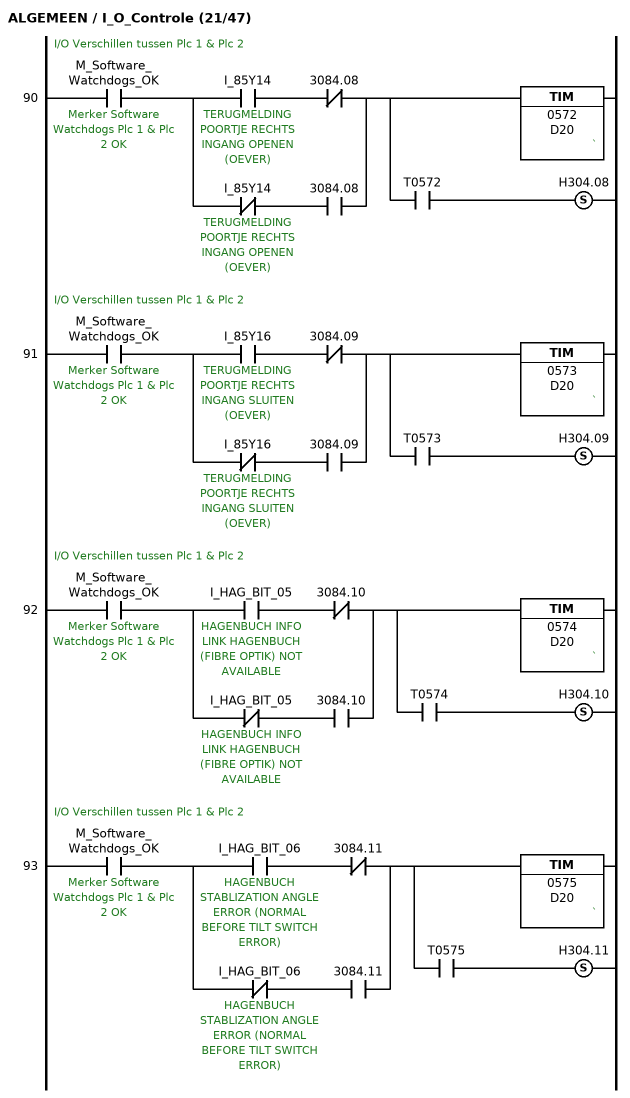
; [picture p229: ALGEMEEN / I_O_Controle, rungs 90-93]
; rung 90: I/O Verschillen tussen Plc 1 & Plc 2
LD M_Software_Watchdogs_OK  ; Merker Software Watchdogs Plc 1 & Plc 2 OK
LD I_85Y14  ; TERUGMELDING POORTJE RECHTS INGANG OPENEN (OEVER)
ANDNOT 3084.08
LDNOT I_85Y14  ; TERUGMELDING POORTJE RECHTS INGANG OPENEN (OEVER)
AND 3084.08
ORLD
ANDLD
TIM 0572 D20  ; `
AND T0572
SET H304.08
; rung 91: I/O Verschillen tussen Plc 1 & Plc 2
LD M_Software_Watchdogs_OK  ; Merker Software Watchdogs Plc 1 & Plc 2 OK
LD I_85Y16  ; TERUGMELDING POORTJE RECHTS INGANG SLUITEN (OEVER)
ANDNOT 3084.09
LDNOT I_85Y16  ; TERUGMELDING POORTJE RECHTS INGANG SLUITEN (OEVER)
AND 3084.09
ORLD
ANDLD
TIM 0573 D20  ; `
AND T0573
SET H304.09
; rung 92: I/O Verschillen tussen Plc 1 & Plc 2
LD M_Software_Watchdogs_OK  ; Merker Software Watchdogs Plc 1 & Plc 2 OK
LD I_HAG_BIT_05  ; HAGENBUCH INFO LINK HAGENBUCH (FIBRE OPTIK) NOT AVAILABLE
ANDNOT 3084.10
LDNOT I_HAG_BIT_05  ; HAGENBUCH INFO LINK HAGENBUCH (FIBRE OPTIK) NOT AVAILABLE
AND 3084.10
ORLD
ANDLD
TIM 0574 D20  ; `
AND T0574
SET H304.10
; rung 93: I/O Verschillen tussen Plc 1 & Plc 2
LD M_Software_Watchdogs_OK  ; Merker Software Watchdogs Plc 1 & Plc 2 OK
LD I_HAG_BIT_06  ; HAGENBUCH STABLIZATION ANGLE ERROR (NORMAL BEFORE TILT SWITCH ERROR)
ANDNOT 3084.11
LDNOT I_HAG_BIT_06  ; HAGENBUCH STABLIZATION ANGLE ERROR (NORMAL BEFORE TILT SWITCH ERROR)
AND 3084.11
ORLD
ANDLD
TIM 0575 D20  ; `
AND T0575
SET H304.11

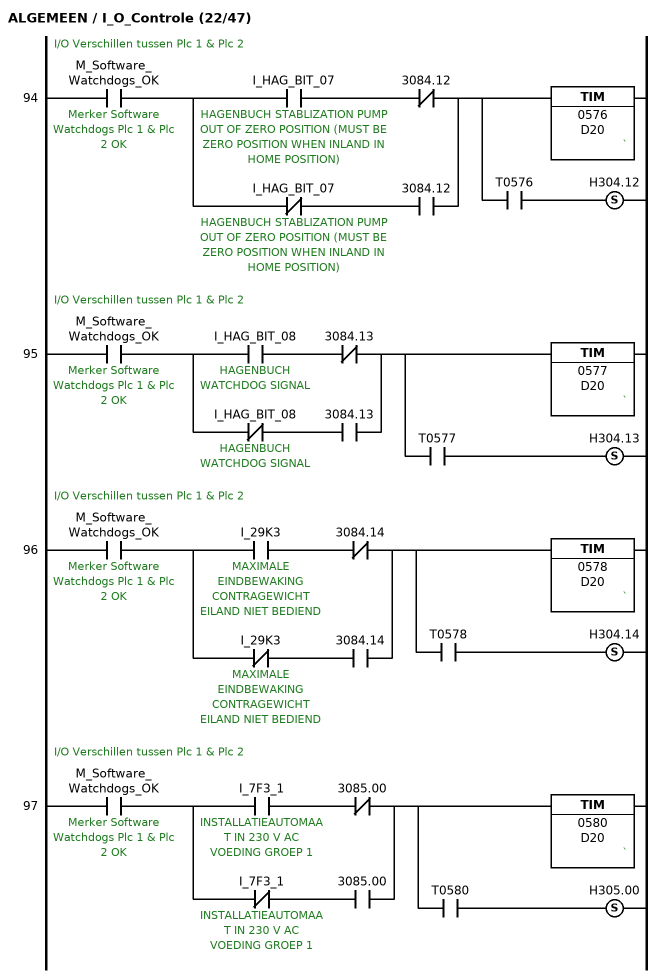
; rung 94: I/O Verschillen tussen Plc 1 & Plc 2
LD M_Software_Watchdogs_OK  ; Merker Software Watchdogs Plc 1 & Plc 2 OK
LD I_HAG_BIT_07  ; HAGENBUCH STABLIZATION PUMP OUT OF ZERO POSITION (MUST BE ZERO POSITION WHEN INLAND IN HOME POSITION)
ANDNOT 3084.12
LDNOT I_HAG_BIT_07  ; HAGENBUCH STABLIZATION PUMP OUT OF ZERO POSITION (MUST BE ZERO POSITION WHEN INLAND IN HOME POSITION)
AND 3084.12
ORLD
ANDLD
TIM 0576 D20  ; `
AND T0576
SET H304.12
; rung 95: I/O Verschillen tussen Plc 1 & Plc 2
LD M_Software_Watchdogs_OK  ; Merker Software Watchdogs Plc 1 & Plc 2 OK
LD I_HAG_BIT_08  ; HAGENBUCH WATCHDOG SIGNAL
ANDNOT 3084.13
LDNOT I_HAG_BIT_08  ; HAGENBUCH WATCHDOG SIGNAL
AND 3084.13
ORLD
ANDLD
TIM 0577 D20  ; `
AND T0577
SET H304.13
; rung 96: I/O Verschillen tussen Plc 1 & Plc 2
LD M_Software_Watchdogs_OK  ; Merker Software Watchdogs Plc 1 & Plc 2 OK
LD I_29K3  ; MAXIMALE EINDBEWAKING CONTRAGEWICHT EILAND NIET BEDIEND
ANDNOT 3084.14
LDNOT I_29K3  ; MAXIMALE EINDBEWAKING CONTRAGEWICHT EILAND NIET BEDIEND
AND 3084.14
ORLD
ANDLD
TIM 0578 D20  ; `
AND T0578
SET H304.14
; rung 97: I/O Verschillen tussen Plc 1 & Plc 2
LD M_Software_Watchdogs_OK  ; Merker Software Watchdogs Plc 1 & Plc 2 OK
LD I_7F3_1  ; INSTALLATIEAUTOMAAT IN 230 V AC VOEDING GROEP 1
ANDNOT 3085.00
LDNOT I_7F3_1  ; INSTALLATIEAUTOMAAT IN 230 V AC VOEDING GROEP 1
AND 3085.00
ORLD
ANDLD
TIM 0580 D20  ; `
AND T0580
SET H305.00

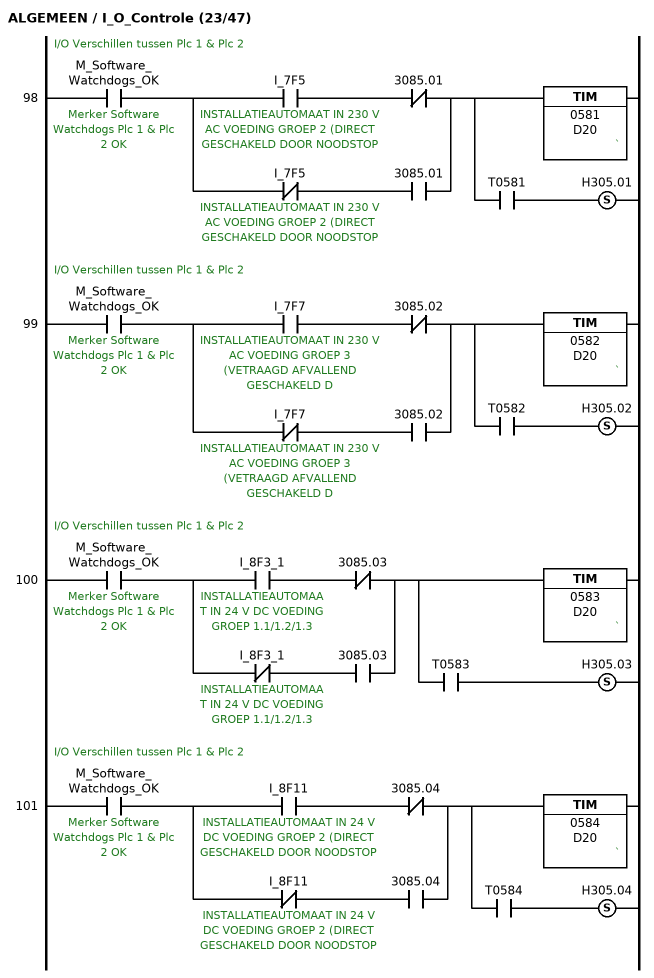
; rung 98: I/O Verschillen tussen Plc 1 & Plc 2
LD M_Software_Watchdogs_OK  ; Merker Software Watchdogs Plc 1 & Plc 2 OK
LD I_7F5  ; INSTALLATIEAUTOMAAT IN 230 V AC VOEDING GROEP 2 (DIRECT GESCHAKELD DOOR NOODSTOP
ANDNOT 3085.01
LDNOT I_7F5  ; INSTALLATIEAUTOMAAT IN 230 V AC VOEDING GROEP 2 (DIRECT GESCHAKELD DOOR NOODSTOP
AND 3085.01
ORLD
ANDLD
TIM 0581 D20  ; `
AND T0581
SET H305.01
; rung 99: I/O Verschillen tussen Plc 1 & Plc 2
LD M_Software_Watchdogs_OK  ; Merker Software Watchdogs Plc 1 & Plc 2 OK
LD I_7F7  ; INSTALLATIEAUTOMAAT IN 230 V AC VOEDING GROEP 3 (VETRAAGD AFVALLEND GESCHAKELD D
ANDNOT 3085.02
LDNOT I_7F7  ; INSTALLATIEAUTOMAAT IN 230 V AC VOEDING GROEP 3 (VETRAAGD AFVALLEND GESCHAKELD D
AND 3085.02
ORLD
ANDLD
TIM 0582 D20  ; `
AND T0582
SET H305.02
; rung 100: I/O Verschillen tussen Plc 1 & Plc 2
LD M_Software_Watchdogs_OK  ; Merker Software Watchdogs Plc 1 & Plc 2 OK
LD I_8F3_1  ; INSTALLATIEAUTOMAAT IN 24 V DC VOEDING GROEP 1.1/1.2/1.3
ANDNOT 3085.03
LDNOT I_8F3_1  ; INSTALLATIEAUTOMAAT IN 24 V DC VOEDING GROEP 1.1/1.2/1.3
AND 3085.03
ORLD
ANDLD
TIM 0583 D20  ; `
AND T0583
SET H305.03
; rung 101: I/O Verschillen tussen Plc 1 & Plc 2
LD M_Software_Watchdogs_OK  ; Merker Software Watchdogs Plc 1 & Plc 2 OK
LD I_8F11  ; INSTALLATIEAUTOMAAT IN 24 V DC VOEDING GROEP 2 (DIRECT GESCHAKELD DOOR NOODSTOP
ANDNOT 3085.04
LDNOT I_8F11  ; INSTALLATIEAUTOMAAT IN 24 V DC VOEDING GROEP 2 (DIRECT GESCHAKELD DOOR NOODSTOP
AND 3085.04
ORLD
ANDLD
TIM 0584 D20  ; `
AND T0584
SET H305.04

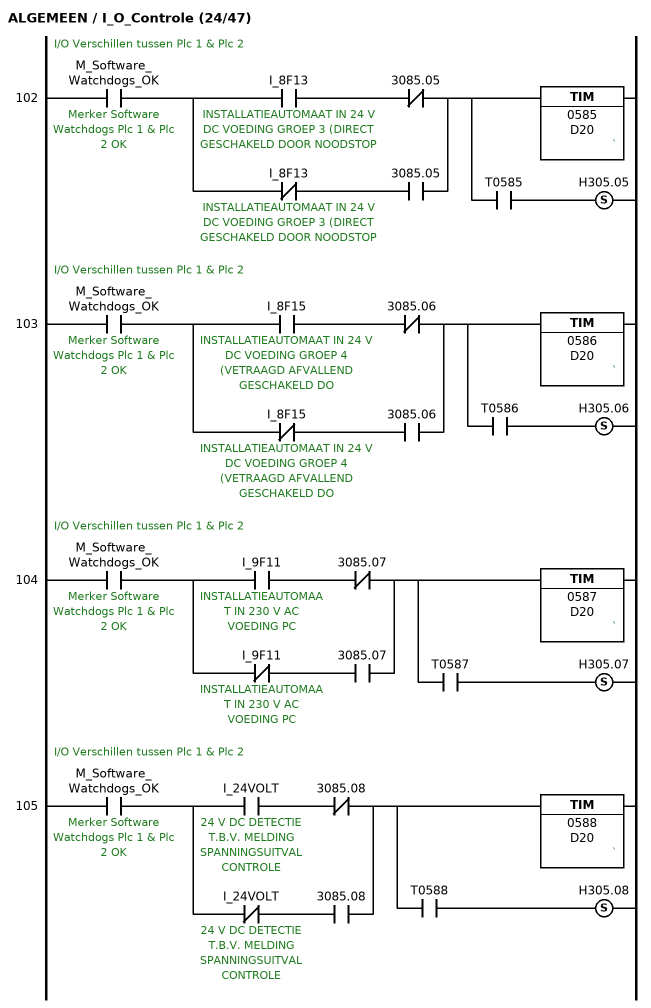
; rung 102: I/O Verschillen tussen Plc 1 & Plc 2
LD M_Software_Watchdogs_OK  ; Merker Software Watchdogs Plc 1 & Plc 2 OK
LD I_8F13  ; INSTALLATIEAUTOMAAT IN 24 V DC VOEDING GROEP 3 (DIRECT GESCHAKELD DOOR NOODSTOP
ANDNOT 3085.05
LDNOT I_8F13  ; INSTALLATIEAUTOMAAT IN 24 V DC VOEDING GROEP 3 (DIRECT GESCHAKELD DOOR NOODSTOP
AND 3085.05
ORLD
ANDLD
TIM 0585 D20  ; `
AND T0585
SET H305.05
; rung 103: I/O Verschillen tussen Plc 1 & Plc 2
LD M_Software_Watchdogs_OK  ; Merker Software Watchdogs Plc 1 & Plc 2 OK
LD I_8F15  ; INSTALLATIEAUTOMAAT IN 24 V DC VOEDING GROEP 4 (VETRAAGD AFVALLEND GESCHAKELD DO
ANDNOT 3085.06
LDNOT I_8F15  ; INSTALLATIEAUTOMAAT IN 24 V DC VOEDING GROEP 4 (VETRAAGD AFVALLEND GESCHAKELD DO
AND 3085.06
ORLD
ANDLD
TIM 0586 D20  ; `
AND T0586
SET H305.06
; rung 104: I/O Verschillen tussen Plc 1 & Plc 2
LD M_Software_Watchdogs_OK  ; Merker Software Watchdogs Plc 1 & Plc 2 OK
LD I_9F11  ; INSTALLATIEAUTOMAAT IN 230 V AC VOEDING PC
ANDNOT 3085.07
LDNOT I_9F11  ; INSTALLATIEAUTOMAAT IN 230 V AC VOEDING PC
AND 3085.07
ORLD
ANDLD
TIM 0587 D20  ; `
AND T0587
SET H305.07
; rung 105: I/O Verschillen tussen Plc 1 & Plc 2
LD M_Software_Watchdogs_OK  ; Merker Software Watchdogs Plc 1 & Plc 2 OK
LD I_24VOLT  ; 24 V DC DETECTIE T.B.V. MELDING SPANNINGSUITVAL CONTROLE
ANDNOT 3085.08
LDNOT I_24VOLT  ; 24 V DC DETECTIE T.B.V. MELDING SPANNINGSUITVAL CONTROLE
AND 3085.08
ORLD
ANDLD
TIM 0588 D20  ; `
AND T0588
SET H305.08

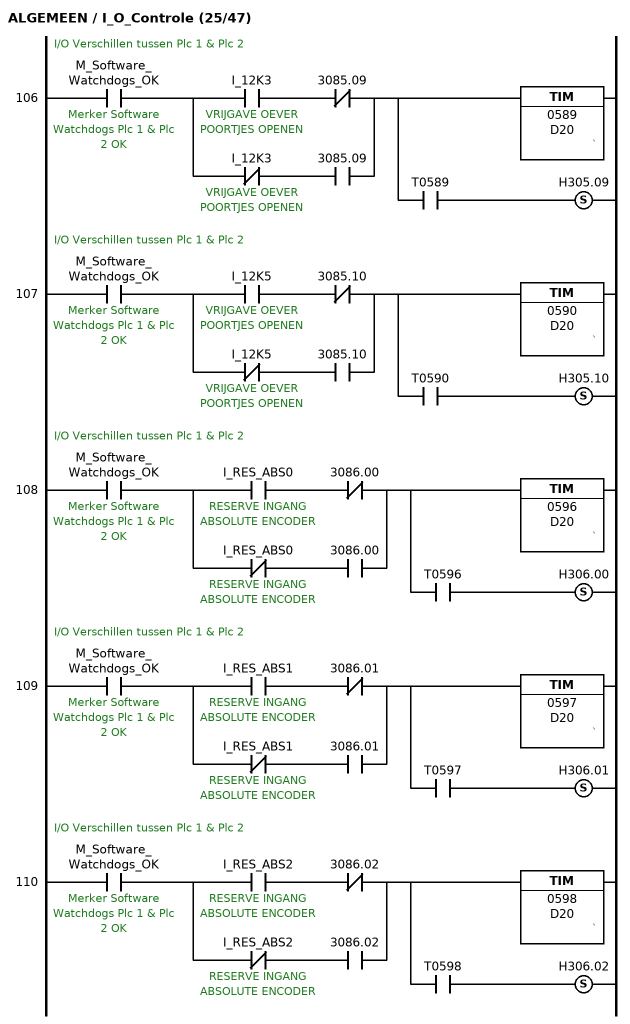
; rung 106: I/O Verschillen tussen Plc 1 & Plc 2
LD M_Software_Watchdogs_OK  ; Merker Software Watchdogs Plc 1 & Plc 2 OK
LD I_12K3  ; VRIJGAVE OEVER POORTJES OPENEN
ANDNOT 3085.09
LDNOT I_12K3  ; VRIJGAVE OEVER POORTJES OPENEN
AND 3085.09
ORLD
ANDLD
TIM 0589 D20  ; `
AND T0589
SET H305.09
; rung 107: I/O Verschillen tussen Plc 1 & Plc 2
LD M_Software_Watchdogs_OK  ; Merker Software Watchdogs Plc 1 & Plc 2 OK
LD I_12K5  ; VRIJGAVE OEVER POORTJES OPENEN
ANDNOT 3085.10
LDNOT I_12K5  ; VRIJGAVE OEVER POORTJES OPENEN
AND 3085.10
ORLD
ANDLD
TIM 0590 D20  ; `
AND T0590
SET H305.10
; rung 108: I/O Verschillen tussen Plc 1 & Plc 2
LD M_Software_Watchdogs_OK  ; Merker Software Watchdogs Plc 1 & Plc 2 OK
LD I_RES_ABS0  ; RESERVE INGANG ABSOLUTE ENCODER
ANDNOT 3086.00
LDNOT I_RES_ABS0  ; RESERVE INGANG ABSOLUTE ENCODER
AND 3086.00
ORLD
ANDLD
TIM 0596 D20  ; `
AND T0596
SET H306.00
; rung 109: I/O Verschillen tussen Plc 1 & Plc 2
LD M_Software_Watchdogs_OK  ; Merker Software Watchdogs Plc 1 & Plc 2 OK
LD I_RES_ABS1  ; RESERVE INGANG ABSOLUTE ENCODER
ANDNOT 3086.01
LDNOT I_RES_ABS1  ; RESERVE INGANG ABSOLUTE ENCODER
AND 3086.01
ORLD
ANDLD
TIM 0597 D20  ; `
AND T0597
SET H306.01
; rung 110: I/O Verschillen tussen Plc 1 & Plc 2
LD M_Software_Watchdogs_OK  ; Merker Software Watchdogs Plc 1 & Plc 2 OK
LD I_RES_ABS2  ; RESERVE INGANG ABSOLUTE ENCODER
ANDNOT 3086.02
LDNOT I_RES_ABS2  ; RESERVE INGANG ABSOLUTE ENCODER
AND 3086.02
ORLD
ANDLD
TIM 0598 D20  ; `
AND T0598
SET H306.02

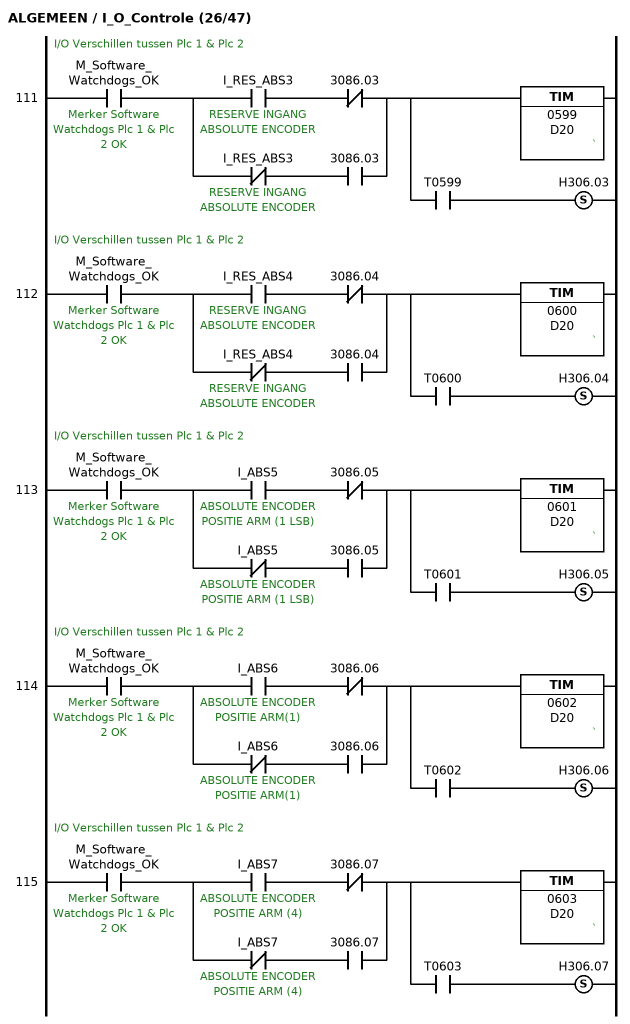
; rung 111: I/O Verschillen tussen Plc 1 & Plc 2
LD M_Software_Watchdogs_OK  ; Merker Software Watchdogs Plc 1 & Plc 2 OK
LD I_RES_ABS3  ; RESERVE INGANG ABSOLUTE ENCODER
ANDNOT 3086.03
LDNOT I_RES_ABS3  ; RESERVE INGANG ABSOLUTE ENCODER
AND 3086.03
ORLD
ANDLD
TIM 0599 D20  ; `
AND T0599
SET H306.03
; rung 112: I/O Verschillen tussen Plc 1 & Plc 2
LD M_Software_Watchdogs_OK  ; Merker Software Watchdogs Plc 1 & Plc 2 OK
LD I_RES_ABS4  ; RESERVE INGANG ABSOLUTE ENCODER
ANDNOT 3086.04
LDNOT I_RES_ABS4  ; RESERVE INGANG ABSOLUTE ENCODER
AND 3086.04
ORLD
ANDLD
TIM 0600 D20  ; `
AND T0600
SET H306.04
; rung 113: I/O Verschillen tussen Plc 1 & Plc 2
LD M_Software_Watchdogs_OK  ; Merker Software Watchdogs Plc 1 & Plc 2 OK
LD I_ABS5  ; ABSOLUTE ENCODER POSITIE ARM (1 LSB)
ANDNOT 3086.05
LDNOT I_ABS5  ; ABSOLUTE ENCODER POSITIE ARM (1 LSB)
AND 3086.05
ORLD
ANDLD
TIM 0601 D20  ; `
AND T0601
SET H306.05
; rung 114: I/O Verschillen tussen Plc 1 & Plc 2
LD M_Software_Watchdogs_OK  ; Merker Software Watchdogs Plc 1 & Plc 2 OK
LD I_ABS6  ; ABSOLUTE ENCODER POSITIE ARM(1)
ANDNOT 3086.06
LDNOT I_ABS6  ; ABSOLUTE ENCODER POSITIE ARM(1)
AND 3086.06
ORLD
ANDLD
TIM 0602 D20  ; `
AND T0602
SET H306.06
; rung 115: I/O Verschillen tussen Plc 1 & Plc 2
LD M_Software_Watchdogs_OK  ; Merker Software Watchdogs Plc 1 & Plc 2 OK
LD I_ABS7  ; ABSOLUTE ENCODER POSITIE ARM (4)
ANDNOT 3086.07
LDNOT I_ABS7  ; ABSOLUTE ENCODER POSITIE ARM (4)
AND 3086.07
ORLD
ANDLD
TIM 0603 D20  ; `
AND T0603
SET H306.07

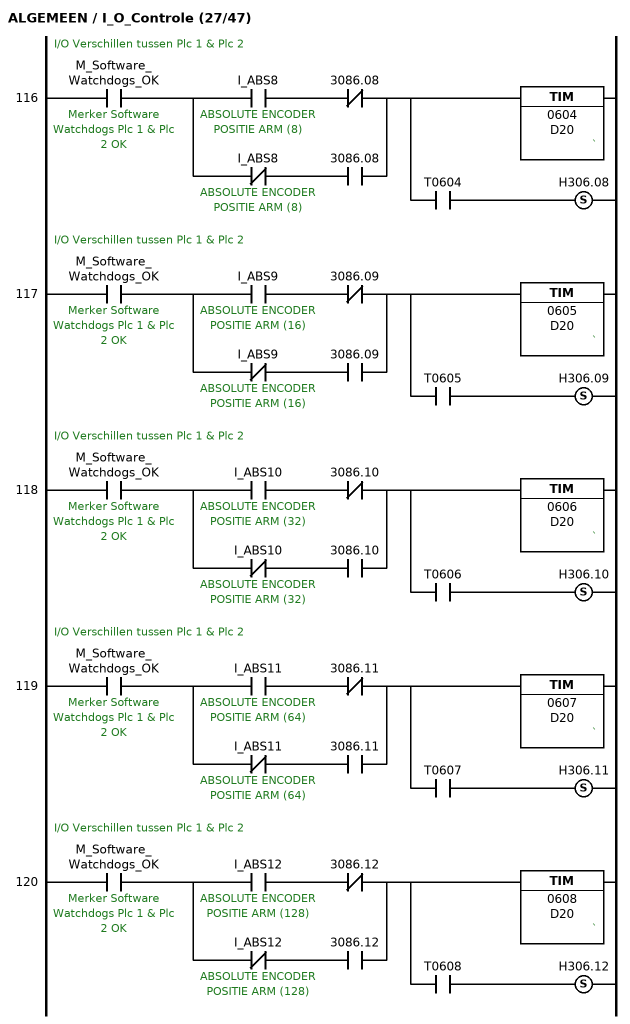
; rung 116: I/O Verschillen tussen Plc 1 & Plc 2
LD M_Software_Watchdogs_OK  ; Merker Software Watchdogs Plc 1 & Plc 2 OK
LD I_ABS8  ; ABSOLUTE ENCODER POSITIE ARM (8)
ANDNOT 3086.08
LDNOT I_ABS8  ; ABSOLUTE ENCODER POSITIE ARM (8)
AND 3086.08
ORLD
ANDLD
TIM 0604 D20  ; `
AND T0604
SET H306.08
; rung 117: I/O Verschillen tussen Plc 1 & Plc 2
LD M_Software_Watchdogs_OK  ; Merker Software Watchdogs Plc 1 & Plc 2 OK
LD I_ABS9  ; ABSOLUTE ENCODER POSITIE ARM (16)
ANDNOT 3086.09
LDNOT I_ABS9  ; ABSOLUTE ENCODER POSITIE ARM (16)
AND 3086.09
ORLD
ANDLD
TIM 0605 D20  ; `
AND T0605
SET H306.09
; rung 118: I/O Verschillen tussen Plc 1 & Plc 2
LD M_Software_Watchdogs_OK  ; Merker Software Watchdogs Plc 1 & Plc 2 OK
LD I_ABS10  ; ABSOLUTE ENCODER POSITIE ARM (32)
ANDNOT 3086.10
LDNOT I_ABS10  ; ABSOLUTE ENCODER POSITIE ARM (32)
AND 3086.10
ORLD
ANDLD
TIM 0606 D20  ; `
AND T0606
SET H306.10
; rung 119: I/O Verschillen tussen Plc 1 & Plc 2
LD M_Software_Watchdogs_OK  ; Merker Software Watchdogs Plc 1 & Plc 2 OK
LD I_ABS11  ; ABSOLUTE ENCODER POSITIE ARM (64)
ANDNOT 3086.11
LDNOT I_ABS11  ; ABSOLUTE ENCODER POSITIE ARM (64)
AND 3086.11
ORLD
ANDLD
TIM 0607 D20  ; `
AND T0607
SET H306.11
; rung 120: I/O Verschillen tussen Plc 1 & Plc 2
LD M_Software_Watchdogs_OK  ; Merker Software Watchdogs Plc 1 & Plc 2 OK
LD I_ABS12  ; ABSOLUTE ENCODER POSITIE ARM (128)
ANDNOT 3086.12
LDNOT I_ABS12  ; ABSOLUTE ENCODER POSITIE ARM (128)
AND 3086.12
ORLD
ANDLD
TIM 0608 D20  ; `
AND T0608
SET H306.12

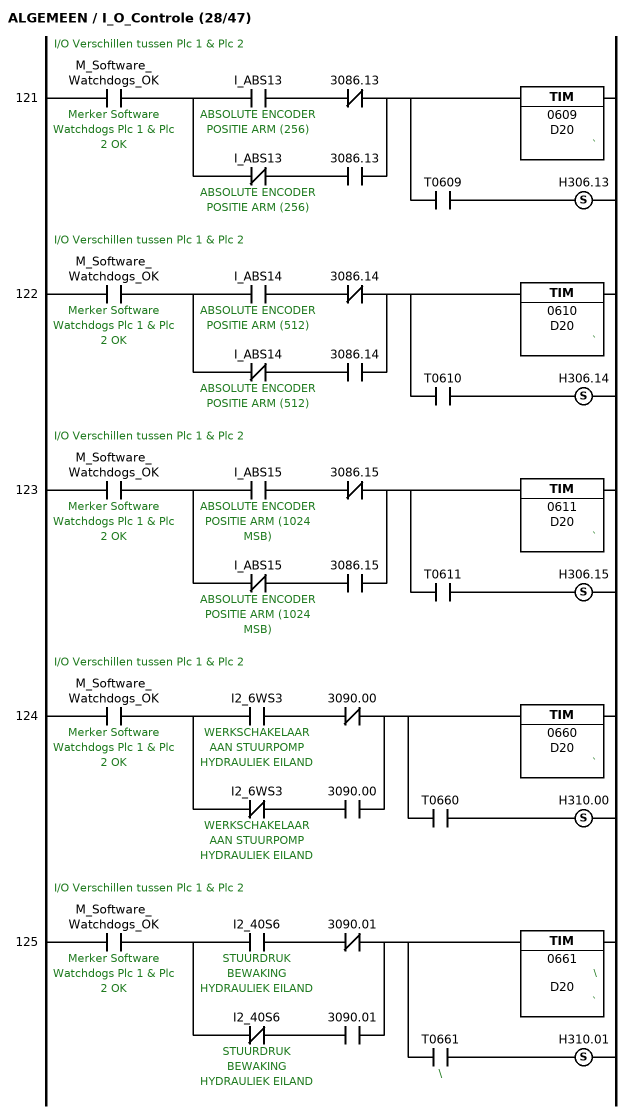
; rung 121: I/O Verschillen tussen Plc 1 & Plc 2
LD M_Software_Watchdogs_OK  ; Merker Software Watchdogs Plc 1 & Plc 2 OK
LD I_ABS13  ; ABSOLUTE ENCODER POSITIE ARM (256)
ANDNOT 3086.13
LDNOT I_ABS13  ; ABSOLUTE ENCODER POSITIE ARM (256)
AND 3086.13
ORLD
ANDLD
TIM 0609 D20  ; `
AND T0609
SET H306.13
; rung 122: I/O Verschillen tussen Plc 1 & Plc 2
LD M_Software_Watchdogs_OK  ; Merker Software Watchdogs Plc 1 & Plc 2 OK
LD I_ABS14  ; ABSOLUTE ENCODER POSITIE ARM (512)
ANDNOT 3086.14
LDNOT I_ABS14  ; ABSOLUTE ENCODER POSITIE ARM (512)
AND 3086.14
ORLD
ANDLD
TIM 0610 D20  ; `
AND T0610
SET H306.14
; rung 123: I/O Verschillen tussen Plc 1 & Plc 2
LD M_Software_Watchdogs_OK  ; Merker Software Watchdogs Plc 1 & Plc 2 OK
LD I_ABS15  ; ABSOLUTE ENCODER POSITIE ARM (1024 MSB)
ANDNOT 3086.15
LDNOT I_ABS15  ; ABSOLUTE ENCODER POSITIE ARM (1024 MSB)
AND 3086.15
ORLD
ANDLD
TIM 0611 D20  ; `
AND T0611
SET H306.15
; rung 124: I/O Verschillen tussen Plc 1 & Plc 2
LD M_Software_Watchdogs_OK  ; Merker Software Watchdogs Plc 1 & Plc 2 OK
LD I2_6WS3  ; WERKSCHAKELAAR AAN STUURPOMP HYDRAULIEK EILAND
ANDNOT 3090.00
LDNOT I2_6WS3  ; WERKSCHAKELAAR AAN STUURPOMP HYDRAULIEK EILAND
AND 3090.00
ORLD
ANDLD
TIM 0660 D20  ; `
AND T0660
SET H310.00
; rung 125: I/O Verschillen tussen Plc 1 & Plc 2
LD M_Software_Watchdogs_OK  ; Merker Software Watchdogs Plc 1 & Plc 2 OK
LD I2_40S6  ; STUURDRUK BEWAKING HYDRAULIEK EILAND
ANDNOT 3090.01
LDNOT I2_40S6  ; STUURDRUK BEWAKING HYDRAULIEK EILAND
AND 3090.01
ORLD
ANDLD
TIM 0661 D20  ; `, \
AND T0661  ; \
SET H310.01

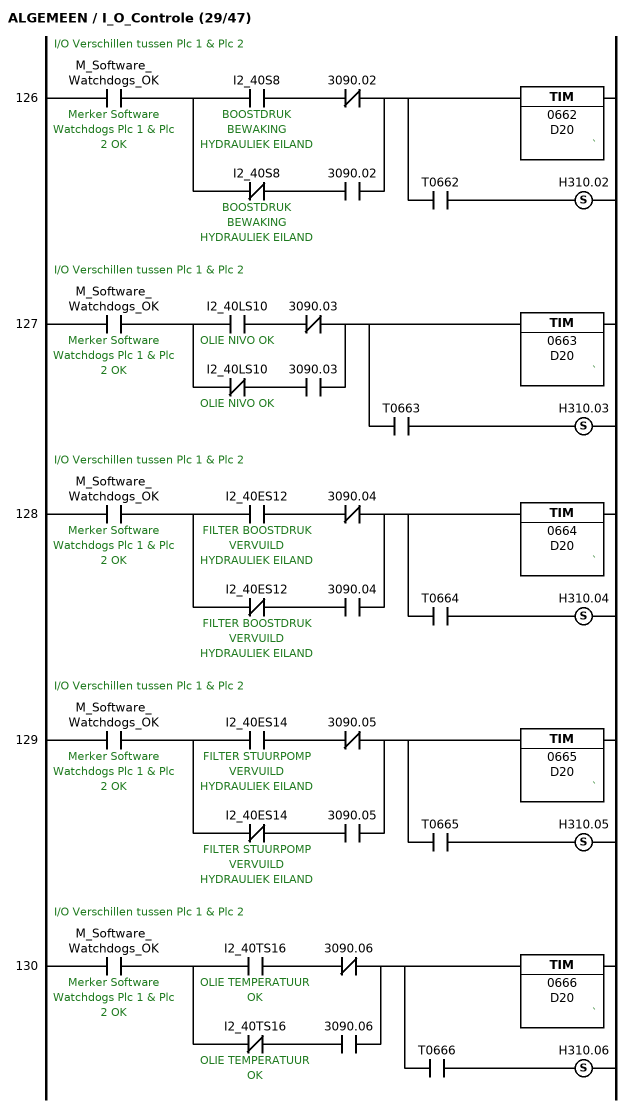
; rung 126: I/O Verschillen tussen Plc 1 & Plc 2
LD M_Software_Watchdogs_OK  ; Merker Software Watchdogs Plc 1 & Plc 2 OK
LD I2_40S8  ; BOOSTDRUK BEWAKING HYDRAULIEK EILAND
ANDNOT 3090.02
LDNOT I2_40S8  ; BOOSTDRUK BEWAKING HYDRAULIEK EILAND
AND 3090.02
ORLD
ANDLD
TIM 0662 D20  ; `
AND T0662
SET H310.02
; rung 127: I/O Verschillen tussen Plc 1 & Plc 2
LD M_Software_Watchdogs_OK  ; Merker Software Watchdogs Plc 1 & Plc 2 OK
LD I2_40LS10  ; OLIE NIVO OK
ANDNOT 3090.03
LDNOT I2_40LS10  ; OLIE NIVO OK
AND 3090.03
ORLD
ANDLD
TIM 0663 D20  ; `
AND T0663
SET H310.03
; rung 128: I/O Verschillen tussen Plc 1 & Plc 2
LD M_Software_Watchdogs_OK  ; Merker Software Watchdogs Plc 1 & Plc 2 OK
LD I2_40ES12  ; FILTER BOOSTDRUK VERVUILD HYDRAULIEK EILAND
ANDNOT 3090.04
LDNOT I2_40ES12  ; FILTER BOOSTDRUK VERVUILD HYDRAULIEK EILAND
AND 3090.04
ORLD
ANDLD
TIM 0664 D20  ; `
AND T0664
SET H310.04
; rung 129: I/O Verschillen tussen Plc 1 & Plc 2
LD M_Software_Watchdogs_OK  ; Merker Software Watchdogs Plc 1 & Plc 2 OK
LD I2_40ES14  ; FILTER STUURPOMP VERVUILD HYDRAULIEK EILAND
ANDNOT 3090.05
LDNOT I2_40ES14  ; FILTER STUURPOMP VERVUILD HYDRAULIEK EILAND
AND 3090.05
ORLD
ANDLD
TIM 0665 D20  ; `
AND T0665
SET H310.05
; rung 130: I/O Verschillen tussen Plc 1 & Plc 2
LD M_Software_Watchdogs_OK  ; Merker Software Watchdogs Plc 1 & Plc 2 OK
LD I2_40TS16  ; OLIE TEMPERATUUR OK
ANDNOT 3090.06
LDNOT I2_40TS16  ; OLIE TEMPERATUUR OK
AND 3090.06
ORLD
ANDLD
TIM 0666 D20  ; `
AND T0666
SET H310.06

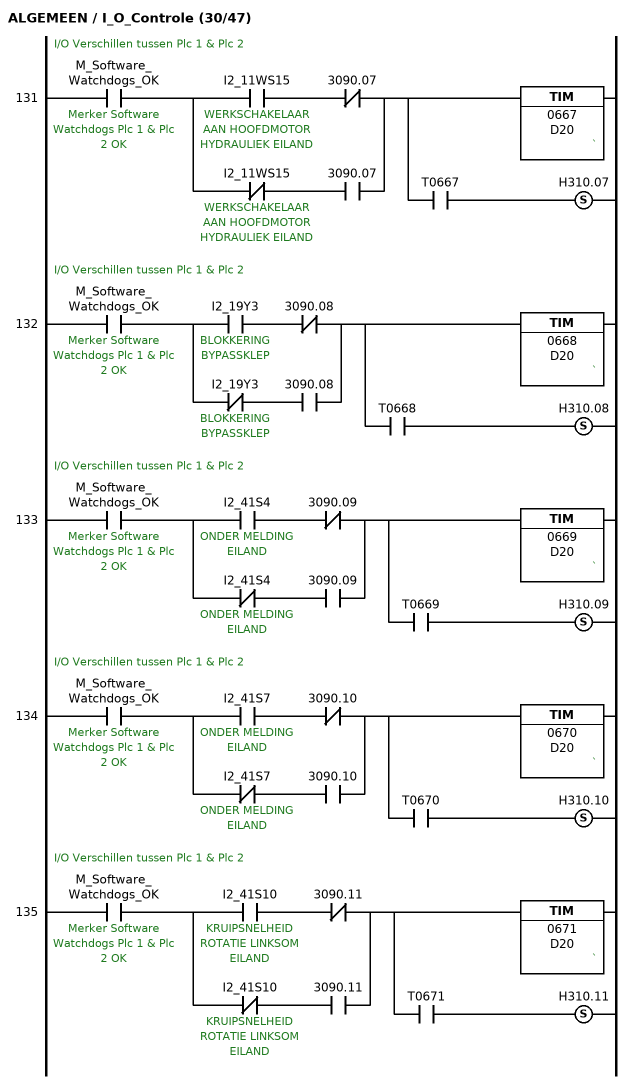
; rung 131: I/O Verschillen tussen Plc 1 & Plc 2
LD M_Software_Watchdogs_OK  ; Merker Software Watchdogs Plc 1 & Plc 2 OK
LD I2_11WS15  ; WERKSCHAKELAAR AAN HOOFDMOTOR HYDRAULIEK EILAND
ANDNOT 3090.07
LDNOT I2_11WS15  ; WERKSCHAKELAAR AAN HOOFDMOTOR HYDRAULIEK EILAND
AND 3090.07
ORLD
ANDLD
TIM 0667 D20  ; `
AND T0667
SET H310.07
; rung 132: I/O Verschillen tussen Plc 1 & Plc 2
LD M_Software_Watchdogs_OK  ; Merker Software Watchdogs Plc 1 & Plc 2 OK
LD I2_19Y3  ; BLOKKERING BYPASSKLEP
ANDNOT 3090.08
LDNOT I2_19Y3  ; BLOKKERING BYPASSKLEP
AND 3090.08
ORLD
ANDLD
TIM 0668 D20  ; `
AND T0668
SET H310.08
; rung 133: I/O Verschillen tussen Plc 1 & Plc 2
LD M_Software_Watchdogs_OK  ; Merker Software Watchdogs Plc 1 & Plc 2 OK
LD I2_41S4  ; ONDER MELDING EILAND
ANDNOT 3090.09
LDNOT I2_41S4  ; ONDER MELDING EILAND
AND 3090.09
ORLD
ANDLD
TIM 0669 D20  ; `
AND T0669
SET H310.09
; rung 134: I/O Verschillen tussen Plc 1 & Plc 2
LD M_Software_Watchdogs_OK  ; Merker Software Watchdogs Plc 1 & Plc 2 OK
LD I2_41S7  ; ONDER MELDING EILAND
ANDNOT 3090.10
LDNOT I2_41S7  ; ONDER MELDING EILAND
AND 3090.10
ORLD
ANDLD
TIM 0670 D20  ; `
AND T0670
SET H310.10
; rung 135: I/O Verschillen tussen Plc 1 & Plc 2
LD M_Software_Watchdogs_OK  ; Merker Software Watchdogs Plc 1 & Plc 2 OK
LD I2_41S10  ; KRUIPSNELHEID ROTATIE LINKSOM EILAND
ANDNOT 3090.11
LDNOT I2_41S10  ; KRUIPSNELHEID ROTATIE LINKSOM EILAND
AND 3090.11
ORLD
ANDLD
TIM 0671 D20  ; `
AND T0671
SET H310.11

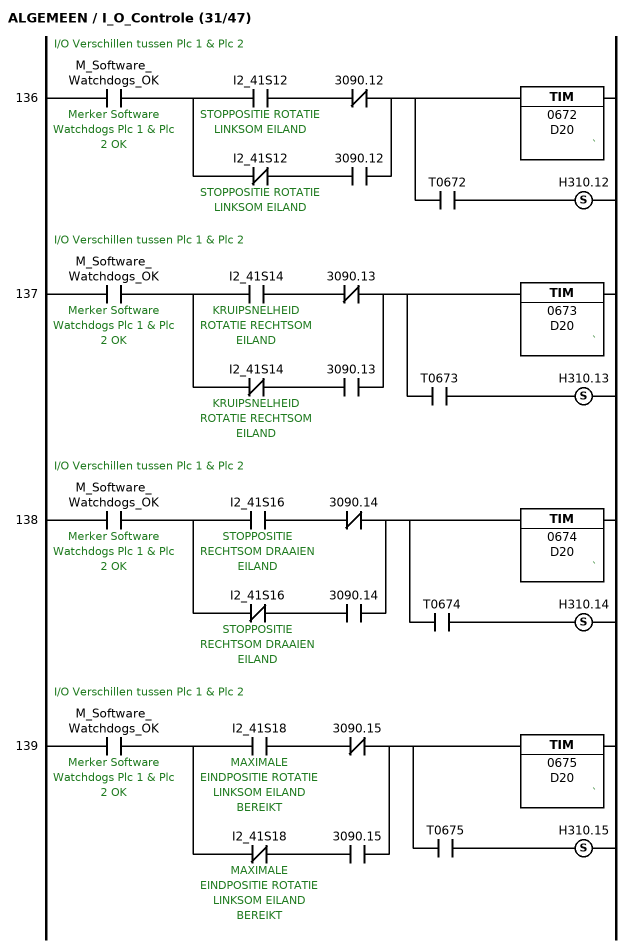
; rung 136: I/O Verschillen tussen Plc 1 & Plc 2
LD M_Software_Watchdogs_OK  ; Merker Software Watchdogs Plc 1 & Plc 2 OK
LD I2_41S12  ; STOPPOSITIE ROTATIE LINKSOM EILAND
ANDNOT 3090.12
LDNOT I2_41S12  ; STOPPOSITIE ROTATIE LINKSOM EILAND
AND 3090.12
ORLD
ANDLD
TIM 0672 D20  ; `
AND T0672
SET H310.12
; rung 137: I/O Verschillen tussen Plc 1 & Plc 2
LD M_Software_Watchdogs_OK  ; Merker Software Watchdogs Plc 1 & Plc 2 OK
LD I2_41S14  ; KRUIPSNELHEID ROTATIE RECHTSOM EILAND
ANDNOT 3090.13
LDNOT I2_41S14  ; KRUIPSNELHEID ROTATIE RECHTSOM EILAND
AND 3090.13
ORLD
ANDLD
TIM 0673 D20  ; `
AND T0673
SET H310.13
; rung 138: I/O Verschillen tussen Plc 1 & Plc 2
LD M_Software_Watchdogs_OK  ; Merker Software Watchdogs Plc 1 & Plc 2 OK
LD I2_41S16  ; STOPPOSITIE RECHTSOM DRAAIEN EILAND
ANDNOT 3090.14
LDNOT I2_41S16  ; STOPPOSITIE RECHTSOM DRAAIEN EILAND
AND 3090.14
ORLD
ANDLD
TIM 0674 D20  ; `
AND T0674
SET H310.14
; rung 139: I/O Verschillen tussen Plc 1 & Plc 2
LD M_Software_Watchdogs_OK  ; Merker Software Watchdogs Plc 1 & Plc 2 OK
LD I2_41S18  ; MAXIMALE EINDPOSITIE ROTATIE LINKSOM EILAND BEREIKT
ANDNOT 3090.15
LDNOT I2_41S18  ; MAXIMALE EINDPOSITIE ROTATIE LINKSOM EILAND BEREIKT
AND 3090.15
ORLD
ANDLD
TIM 0675 D20  ; `
AND T0675
SET H310.15

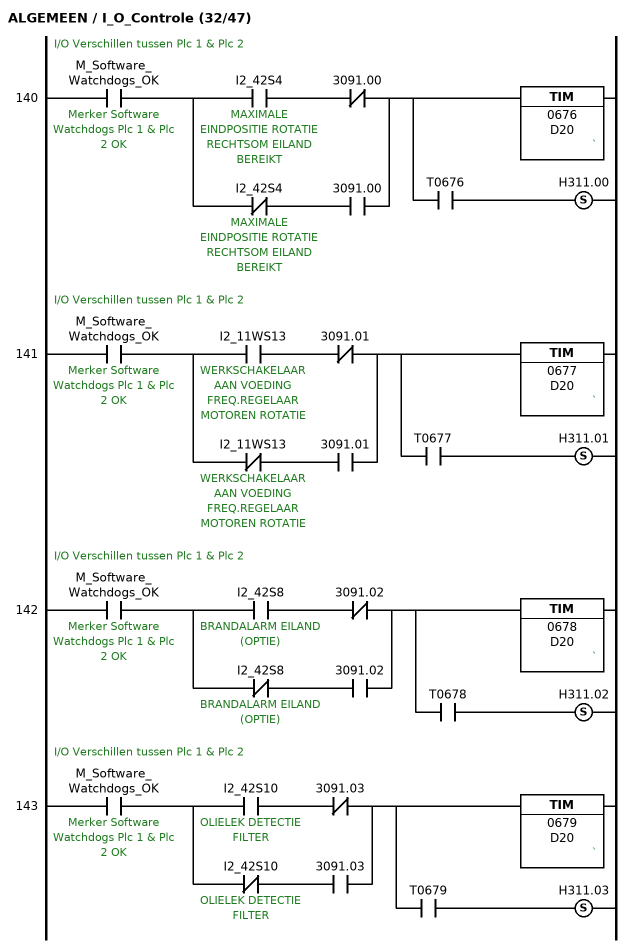
; rung 140: I/O Verschillen tussen Plc 1 & Plc 2
LD M_Software_Watchdogs_OK  ; Merker Software Watchdogs Plc 1 & Plc 2 OK
LD I2_42S4  ; MAXIMALE EINDPOSITIE ROTATIE RECHTSOM EILAND BEREIKT
ANDNOT 3091.00
LDNOT I2_42S4  ; MAXIMALE EINDPOSITIE ROTATIE RECHTSOM EILAND BEREIKT
AND 3091.00
ORLD
ANDLD
TIM 0676 D20  ; `
AND T0676
SET H311.00
; rung 141: I/O Verschillen tussen Plc 1 & Plc 2
LD M_Software_Watchdogs_OK  ; Merker Software Watchdogs Plc 1 & Plc 2 OK
LD I2_11WS13  ; WERKSCHAKELAAR AAN VOEDING FREQ.REGELAAR MOTOREN ROTATIE
ANDNOT 3091.01
LDNOT I2_11WS13  ; WERKSCHAKELAAR AAN VOEDING FREQ.REGELAAR MOTOREN ROTATIE
AND 3091.01
ORLD
ANDLD
TIM 0677 D20  ; `
AND T0677
SET H311.01
; rung 142: I/O Verschillen tussen Plc 1 & Plc 2
LD M_Software_Watchdogs_OK  ; Merker Software Watchdogs Plc 1 & Plc 2 OK
LD I2_42S8  ; BRANDALARM EILAND (OPTIE)
ANDNOT 3091.02
LDNOT I2_42S8  ; BRANDALARM EILAND (OPTIE)
AND 3091.02
ORLD
ANDLD
TIM 0678 D20  ; `
AND T0678
SET H311.02
; rung 143: I/O Verschillen tussen Plc 1 & Plc 2
LD M_Software_Watchdogs_OK  ; Merker Software Watchdogs Plc 1 & Plc 2 OK
LD I2_42S10  ; OLIELEK DETECTIE FILTER
ANDNOT 3091.03
LDNOT I2_42S10  ; OLIELEK DETECTIE FILTER
AND 3091.03
ORLD
ANDLD
TIM 0679 D20  ; `
AND T0679
SET H311.03

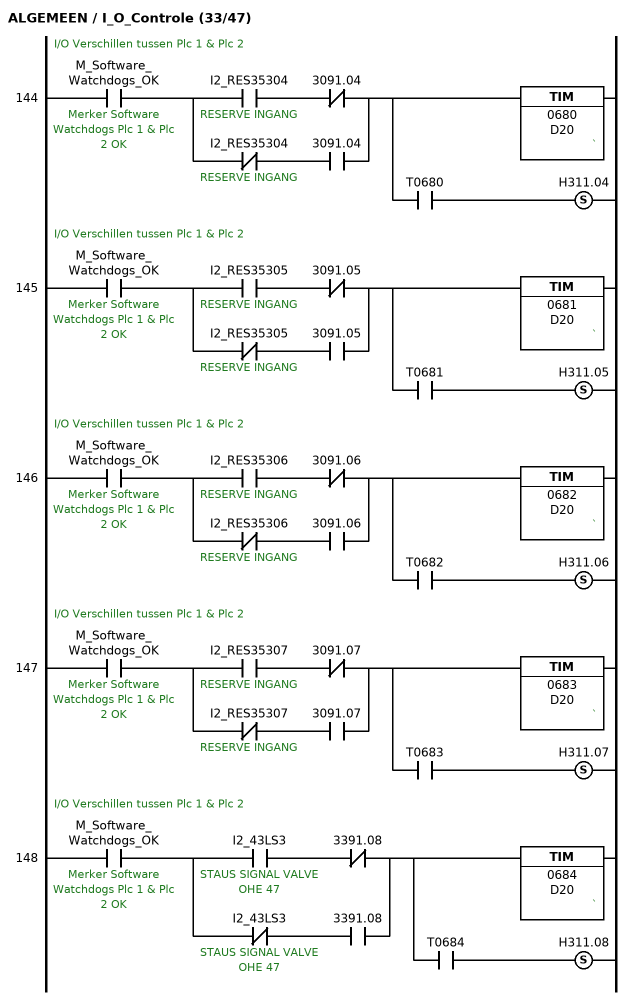
; rung 144: I/O Verschillen tussen Plc 1 & Plc 2
LD M_Software_Watchdogs_OK  ; Merker Software Watchdogs Plc 1 & Plc 2 OK
LD I2_RES35304  ; RESERVE INGANG
ANDNOT 3091.04
LDNOT I2_RES35304  ; RESERVE INGANG
AND 3091.04
ORLD
ANDLD
TIM 0680 D20  ; `
AND T0680
SET H311.04
; rung 145: I/O Verschillen tussen Plc 1 & Plc 2
LD M_Software_Watchdogs_OK  ; Merker Software Watchdogs Plc 1 & Plc 2 OK
LD I2_RES35305  ; RESERVE INGANG
ANDNOT 3091.05
LDNOT I2_RES35305  ; RESERVE INGANG
AND 3091.05
ORLD
ANDLD
TIM 0681 D20  ; `
AND T0681
SET H311.05
; rung 146: I/O Verschillen tussen Plc 1 & Plc 2
LD M_Software_Watchdogs_OK  ; Merker Software Watchdogs Plc 1 & Plc 2 OK
LD I2_RES35306  ; RESERVE INGANG
ANDNOT 3091.06
LDNOT I2_RES35306  ; RESERVE INGANG
AND 3091.06
ORLD
ANDLD
TIM 0682 D20  ; `
AND T0682
SET H311.06
; rung 147: I/O Verschillen tussen Plc 1 & Plc 2
LD M_Software_Watchdogs_OK  ; Merker Software Watchdogs Plc 1 & Plc 2 OK
LD I2_RES35307  ; RESERVE INGANG
ANDNOT 3091.07
LDNOT I2_RES35307  ; RESERVE INGANG
AND 3091.07
ORLD
ANDLD
TIM 0683 D20  ; `
AND T0683
SET H311.07
; rung 148: I/O Verschillen tussen Plc 1 & Plc 2
LD M_Software_Watchdogs_OK  ; Merker Software Watchdogs Plc 1 & Plc 2 OK
LD I2_43LS3  ; STAUS SIGNAL VALVE OHE 47
ANDNOT 3391.08
LDNOT I2_43LS3  ; STAUS SIGNAL VALVE OHE 47
AND 3391.08
ORLD
ANDLD
TIM 0684 D20  ; `
AND T0684
SET H311.08

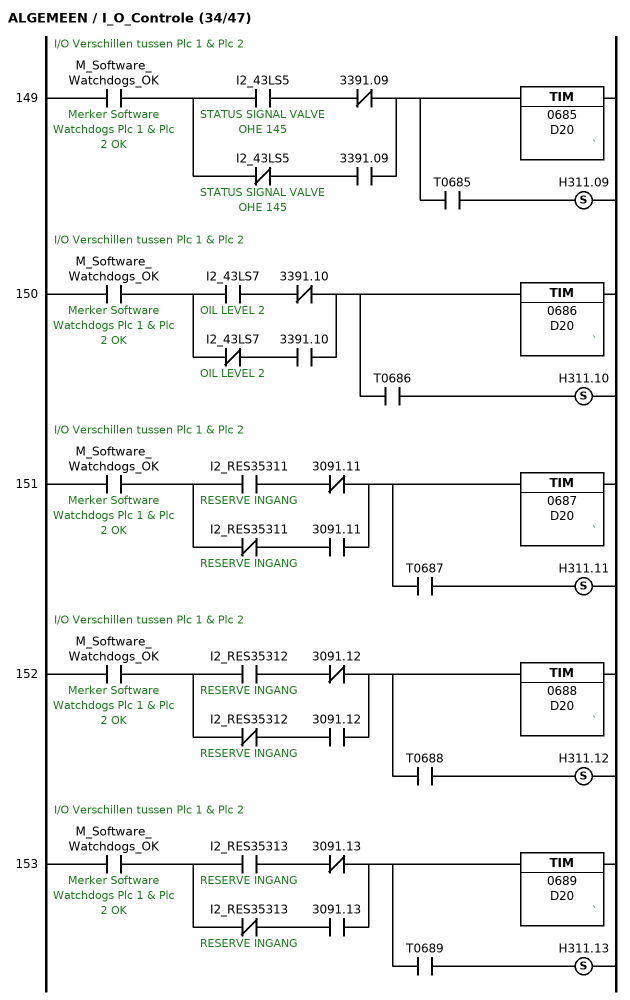
; rung 149: I/O Verschillen tussen Plc 1 & Plc 2
LD M_Software_Watchdogs_OK  ; Merker Software Watchdogs Plc 1 & Plc 2 OK
LD I2_43LS5  ; STATUS SIGNAL VALVE OHE 145
ANDNOT 3391.09
LDNOT I2_43LS5  ; STATUS SIGNAL VALVE OHE 145
AND 3391.09
ORLD
ANDLD
TIM 0685 D20  ; `
AND T0685
SET H311.09
; rung 150: I/O Verschillen tussen Plc 1 & Plc 2
LD M_Software_Watchdogs_OK  ; Merker Software Watchdogs Plc 1 & Plc 2 OK
LD I2_43LS7  ; OIL LEVEL 2
ANDNOT 3391.10
LDNOT I2_43LS7  ; OIL LEVEL 2
AND 3391.10
ORLD
ANDLD
TIM 0686 D20  ; `
AND T0686
SET H311.10
; rung 151: I/O Verschillen tussen Plc 1 & Plc 2
LD M_Software_Watchdogs_OK  ; Merker Software Watchdogs Plc 1 & Plc 2 OK
LD I2_RES35311  ; RESERVE INGANG
ANDNOT 3091.11
LDNOT I2_RES35311  ; RESERVE INGANG
AND 3091.11
ORLD
ANDLD
TIM 0687 D20  ; `
AND T0687
SET H311.11
; rung 152: I/O Verschillen tussen Plc 1 & Plc 2
LD M_Software_Watchdogs_OK  ; Merker Software Watchdogs Plc 1 & Plc 2 OK
LD I2_RES35312  ; RESERVE INGANG
ANDNOT 3091.12
LDNOT I2_RES35312  ; RESERVE INGANG
AND 3091.12
ORLD
ANDLD
TIM 0688 D20  ; `
AND T0688
SET H311.12
; rung 153: I/O Verschillen tussen Plc 1 & Plc 2
LD M_Software_Watchdogs_OK  ; Merker Software Watchdogs Plc 1 & Plc 2 OK
LD I2_RES35313  ; RESERVE INGANG
ANDNOT 3091.13
LDNOT I2_RES35313  ; RESERVE INGANG
AND 3091.13
ORLD
ANDLD
TIM 0689 D20  ; `
AND T0689
SET H311.13

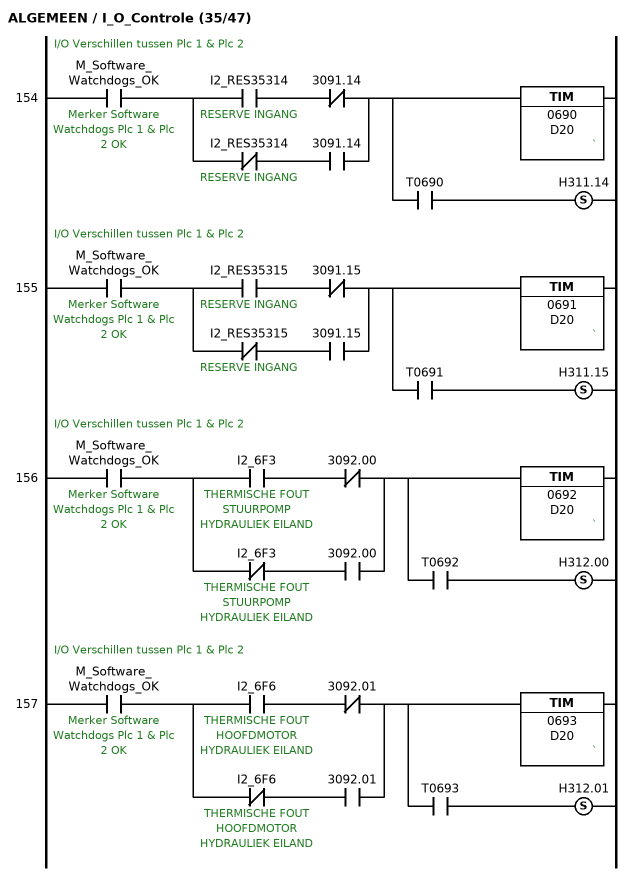
; rung 154: I/O Verschillen tussen Plc 1 & Plc 2
LD M_Software_Watchdogs_OK  ; Merker Software Watchdogs Plc 1 & Plc 2 OK
LD I2_RES35314  ; RESERVE INGANG
ANDNOT 3091.14
LDNOT I2_RES35314  ; RESERVE INGANG
AND 3091.14
ORLD
ANDLD
TIM 0690 D20  ; `
AND T0690
SET H311.14
; rung 155: I/O Verschillen tussen Plc 1 & Plc 2
LD M_Software_Watchdogs_OK  ; Merker Software Watchdogs Plc 1 & Plc 2 OK
LD I2_RES35315  ; RESERVE INGANG
ANDNOT 3091.15
LDNOT I2_RES35315  ; RESERVE INGANG
AND 3091.15
ORLD
ANDLD
TIM 0691 D20  ; `
AND T0691
SET H311.15
; rung 156: I/O Verschillen tussen Plc 1 & Plc 2
LD M_Software_Watchdogs_OK  ; Merker Software Watchdogs Plc 1 & Plc 2 OK
LD I2_6F3  ; THERMISCHE FOUT STUURPOMP HYDRAULIEK EILAND
ANDNOT 3092.00
LDNOT I2_6F3  ; THERMISCHE FOUT STUURPOMP HYDRAULIEK EILAND
AND 3092.00
ORLD
ANDLD
TIM 0692 D20  ; `
AND T0692
SET H312.00
; rung 157: I/O Verschillen tussen Plc 1 & Plc 2
LD M_Software_Watchdogs_OK  ; Merker Software Watchdogs Plc 1 & Plc 2 OK
LD I2_6F6  ; THERMISCHE FOUT HOOFDMOTOR HYDRAULIEK EILAND
ANDNOT 3092.01
LDNOT I2_6F6  ; THERMISCHE FOUT HOOFDMOTOR HYDRAULIEK EILAND
AND 3092.01
ORLD
ANDLD
TIM 0693 D20  ; `
AND T0693
SET H312.01

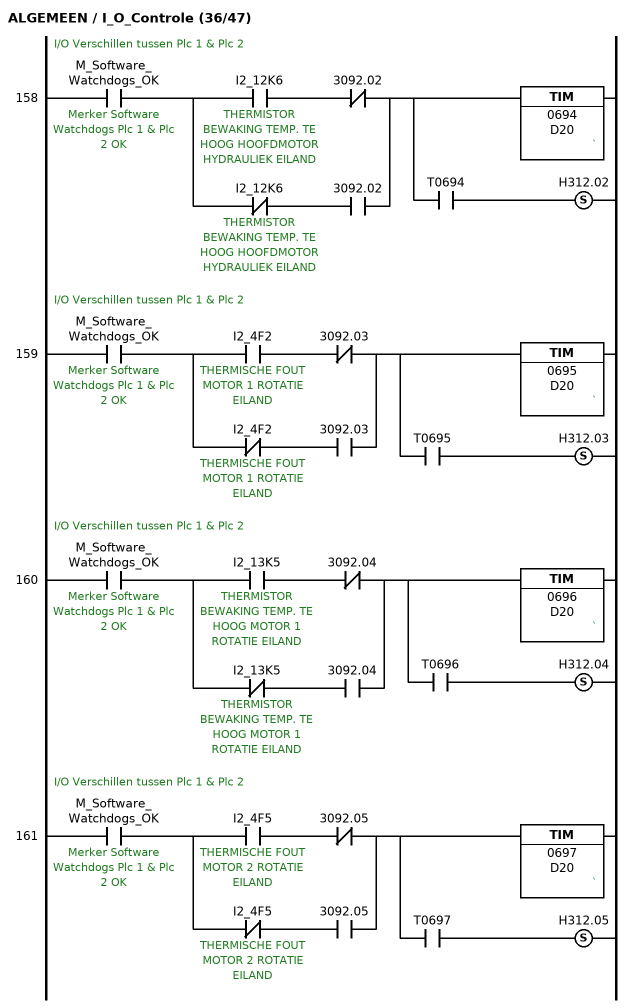
; rung 158: I/O Verschillen tussen Plc 1 & Plc 2
LD M_Software_Watchdogs_OK  ; Merker Software Watchdogs Plc 1 & Plc 2 OK
LD I2_12K6  ; THERMISTOR BEWAKING TEMP. TE HOOG HOOFDMOTOR HYDRAULIEK EILAND
ANDNOT 3092.02
LDNOT I2_12K6  ; THERMISTOR BEWAKING TEMP. TE HOOG HOOFDMOTOR HYDRAULIEK EILAND
AND 3092.02
ORLD
ANDLD
TIM 0694 D20  ; `
AND T0694
SET H312.02
; rung 159: I/O Verschillen tussen Plc 1 & Plc 2
LD M_Software_Watchdogs_OK  ; Merker Software Watchdogs Plc 1 & Plc 2 OK
LD I2_4F2  ; THERMISCHE FOUT MOTOR 1 ROTATIE EILAND
ANDNOT 3092.03
LDNOT I2_4F2  ; THERMISCHE FOUT MOTOR 1 ROTATIE EILAND
AND 3092.03
ORLD
ANDLD
TIM 0695 D20  ; `
AND T0695
SET H312.03
; rung 160: I/O Verschillen tussen Plc 1 & Plc 2
LD M_Software_Watchdogs_OK  ; Merker Software Watchdogs Plc 1 & Plc 2 OK
LD I2_13K5  ; THERMISTOR BEWAKING TEMP. TE HOOG MOTOR 1 ROTATIE EILAND
ANDNOT 3092.04
LDNOT I2_13K5  ; THERMISTOR BEWAKING TEMP. TE HOOG MOTOR 1 ROTATIE EILAND
AND 3092.04
ORLD
ANDLD
TIM 0696 D20  ; `
AND T0696
SET H312.04
; rung 161: I/O Verschillen tussen Plc 1 & Plc 2
LD M_Software_Watchdogs_OK  ; Merker Software Watchdogs Plc 1 & Plc 2 OK
LD I2_4F5  ; THERMISCHE FOUT MOTOR 2 ROTATIE EILAND
ANDNOT 3092.05
LDNOT I2_4F5  ; THERMISCHE FOUT MOTOR 2 ROTATIE EILAND
AND 3092.05
ORLD
ANDLD
TIM 0697 D20  ; `
AND T0697
SET H312.05

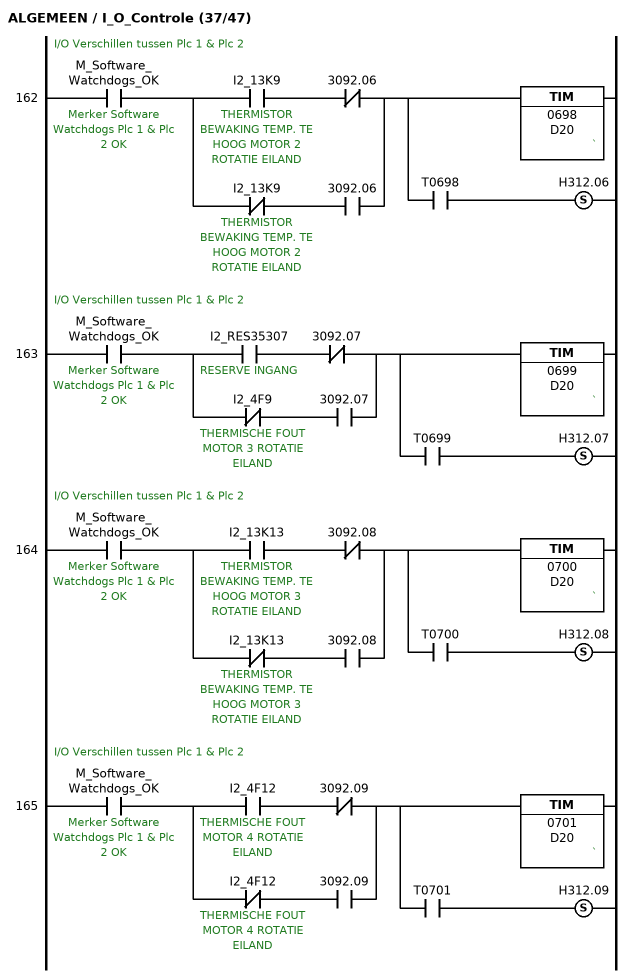
; rung 162: I/O Verschillen tussen Plc 1 & Plc 2
LD M_Software_Watchdogs_OK  ; Merker Software Watchdogs Plc 1 & Plc 2 OK
LD I2_13K9  ; THERMISTOR BEWAKING TEMP. TE HOOG MOTOR 2 ROTATIE EILAND
ANDNOT 3092.06
LDNOT I2_13K9  ; THERMISTOR BEWAKING TEMP. TE HOOG MOTOR 2 ROTATIE EILAND
AND 3092.06
ORLD
ANDLD
TIM 0698 D20  ; `
AND T0698
SET H312.06
; rung 163: I/O Verschillen tussen Plc 1 & Plc 2
LD M_Software_Watchdogs_OK  ; Merker Software Watchdogs Plc 1 & Plc 2 OK
LD I2_RES35307  ; RESERVE INGANG
ANDNOT 3092.07
LDNOT I2_4F9  ; THERMISCHE FOUT MOTOR 3 ROTATIE EILAND
AND 3092.07
ORLD
ANDLD
TIM 0699 D20  ; `
AND T0699
SET H312.07
; rung 164: I/O Verschillen tussen Plc 1 & Plc 2
LD M_Software_Watchdogs_OK  ; Merker Software Watchdogs Plc 1 & Plc 2 OK
LD I2_13K13  ; THERMISTOR BEWAKING TEMP. TE HOOG MOTOR 3 ROTATIE EILAND
ANDNOT 3092.08
LDNOT I2_13K13  ; THERMISTOR BEWAKING TEMP. TE HOOG MOTOR 3 ROTATIE EILAND
AND 3092.08
ORLD
ANDLD
TIM 0700 D20  ; `
AND T0700
SET H312.08
; rung 165: I/O Verschillen tussen Plc 1 & Plc 2
LD M_Software_Watchdogs_OK  ; Merker Software Watchdogs Plc 1 & Plc 2 OK
LD I2_4F12  ; THERMISCHE FOUT MOTOR 4 ROTATIE EILAND
ANDNOT 3092.09
LDNOT I2_4F12  ; THERMISCHE FOUT MOTOR 4 ROTATIE EILAND
AND 3092.09
ORLD
ANDLD
TIM 0701 D20  ; `
AND T0701
SET H312.09

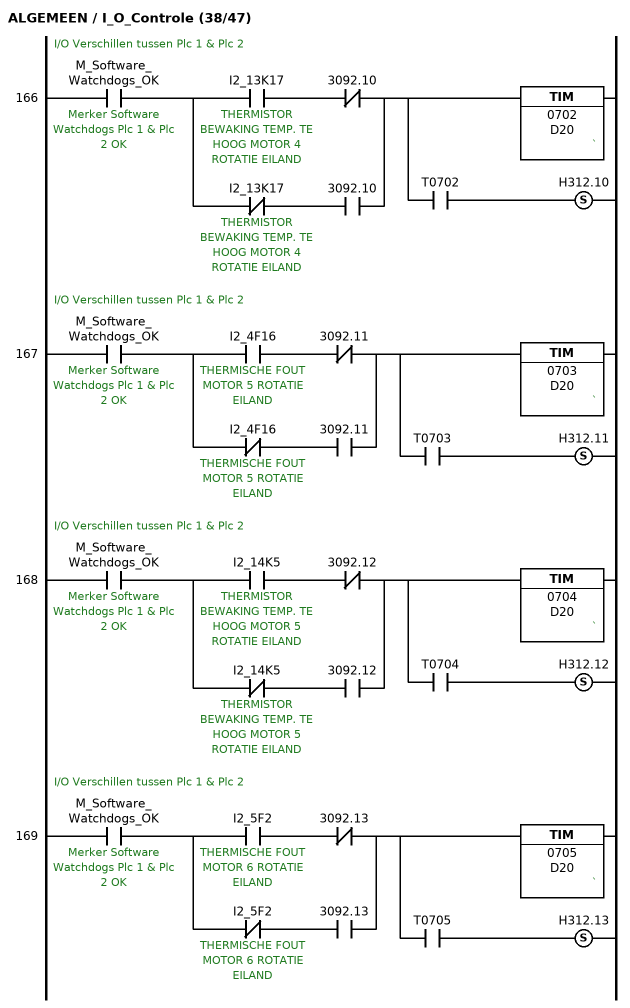
; rung 166: I/O Verschillen tussen Plc 1 & Plc 2
LD M_Software_Watchdogs_OK  ; Merker Software Watchdogs Plc 1 & Plc 2 OK
LD I2_13K17  ; THERMISTOR BEWAKING TEMP. TE HOOG MOTOR 4 ROTATIE EILAND
ANDNOT 3092.10
LDNOT I2_13K17  ; THERMISTOR BEWAKING TEMP. TE HOOG MOTOR 4 ROTATIE EILAND
AND 3092.10
ORLD
ANDLD
TIM 0702 D20  ; `
AND T0702
SET H312.10
; rung 167: I/O Verschillen tussen Plc 1 & Plc 2
LD M_Software_Watchdogs_OK  ; Merker Software Watchdogs Plc 1 & Plc 2 OK
LD I2_4F16  ; THERMISCHE FOUT MOTOR 5 ROTATIE EILAND
ANDNOT 3092.11
LDNOT I2_4F16  ; THERMISCHE FOUT MOTOR 5 ROTATIE EILAND
AND 3092.11
ORLD
ANDLD
TIM 0703 D20  ; `
AND T0703
SET H312.11
; rung 168: I/O Verschillen tussen Plc 1 & Plc 2
LD M_Software_Watchdogs_OK  ; Merker Software Watchdogs Plc 1 & Plc 2 OK
LD I2_14K5  ; THERMISTOR BEWAKING TEMP. TE HOOG MOTOR 5 ROTATIE EILAND
ANDNOT 3092.12
LDNOT I2_14K5  ; THERMISTOR BEWAKING TEMP. TE HOOG MOTOR 5 ROTATIE EILAND
AND 3092.12
ORLD
ANDLD
TIM 0704 D20  ; `
AND T0704
SET H312.12
; rung 169: I/O Verschillen tussen Plc 1 & Plc 2
LD M_Software_Watchdogs_OK  ; Merker Software Watchdogs Plc 1 & Plc 2 OK
LD I2_5F2  ; THERMISCHE FOUT MOTOR 6 ROTATIE EILAND
ANDNOT 3092.13
LDNOT I2_5F2  ; THERMISCHE FOUT MOTOR 6 ROTATIE EILAND
AND 3092.13
ORLD
ANDLD
TIM 0705 D20  ; `
AND T0705
SET H312.13

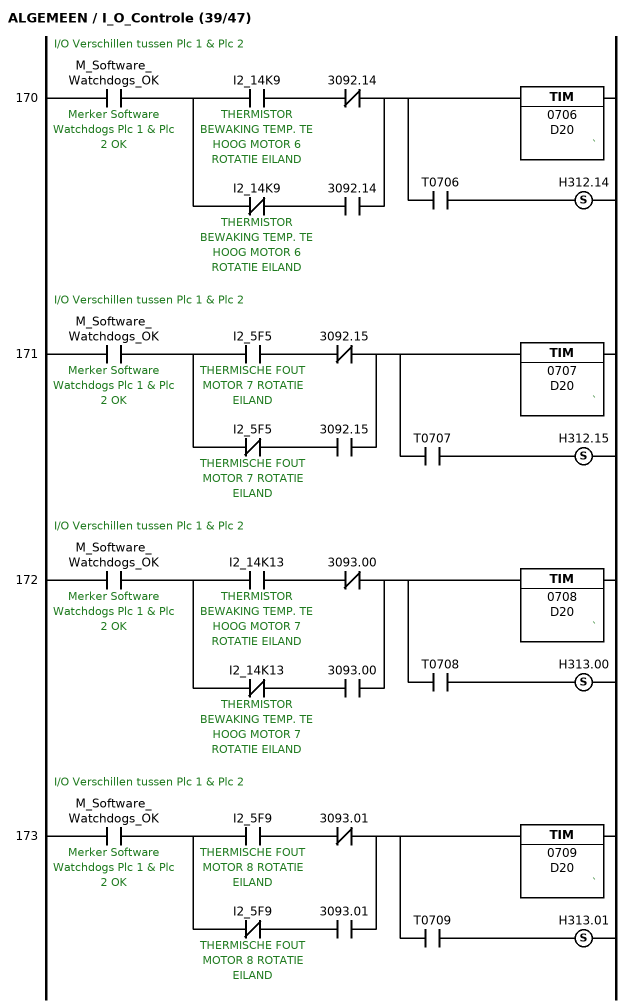
; rung 170: I/O Verschillen tussen Plc 1 & Plc 2
LD M_Software_Watchdogs_OK  ; Merker Software Watchdogs Plc 1 & Plc 2 OK
LD I2_14K9  ; THERMISTOR BEWAKING TEMP. TE HOOG MOTOR 6 ROTATIE EILAND
ANDNOT 3092.14
LDNOT I2_14K9  ; THERMISTOR BEWAKING TEMP. TE HOOG MOTOR 6 ROTATIE EILAND
AND 3092.14
ORLD
ANDLD
TIM 0706 D20  ; `
AND T0706
SET H312.14
; rung 171: I/O Verschillen tussen Plc 1 & Plc 2
LD M_Software_Watchdogs_OK  ; Merker Software Watchdogs Plc 1 & Plc 2 OK
LD I2_5F5  ; THERMISCHE FOUT MOTOR 7 ROTATIE EILAND
ANDNOT 3092.15
LDNOT I2_5F5  ; THERMISCHE FOUT MOTOR 7 ROTATIE EILAND
AND 3092.15
ORLD
ANDLD
TIM 0707 D20  ; `
AND T0707
SET H312.15
; rung 172: I/O Verschillen tussen Plc 1 & Plc 2
LD M_Software_Watchdogs_OK  ; Merker Software Watchdogs Plc 1 & Plc 2 OK
LD I2_14K13  ; THERMISTOR BEWAKING TEMP. TE HOOG MOTOR 7 ROTATIE EILAND
ANDNOT 3093.00
LDNOT I2_14K13  ; THERMISTOR BEWAKING TEMP. TE HOOG MOTOR 7 ROTATIE EILAND
AND 3093.00
ORLD
ANDLD
TIM 0708 D20  ; `
AND T0708
SET H313.00
; rung 173: I/O Verschillen tussen Plc 1 & Plc 2
LD M_Software_Watchdogs_OK  ; Merker Software Watchdogs Plc 1 & Plc 2 OK
LD I2_5F9  ; THERMISCHE FOUT MOTOR 8 ROTATIE EILAND
ANDNOT 3093.01
LDNOT I2_5F9  ; THERMISCHE FOUT MOTOR 8 ROTATIE EILAND
AND 3093.01
ORLD
ANDLD
TIM 0709 D20  ; `
AND T0709
SET H313.01

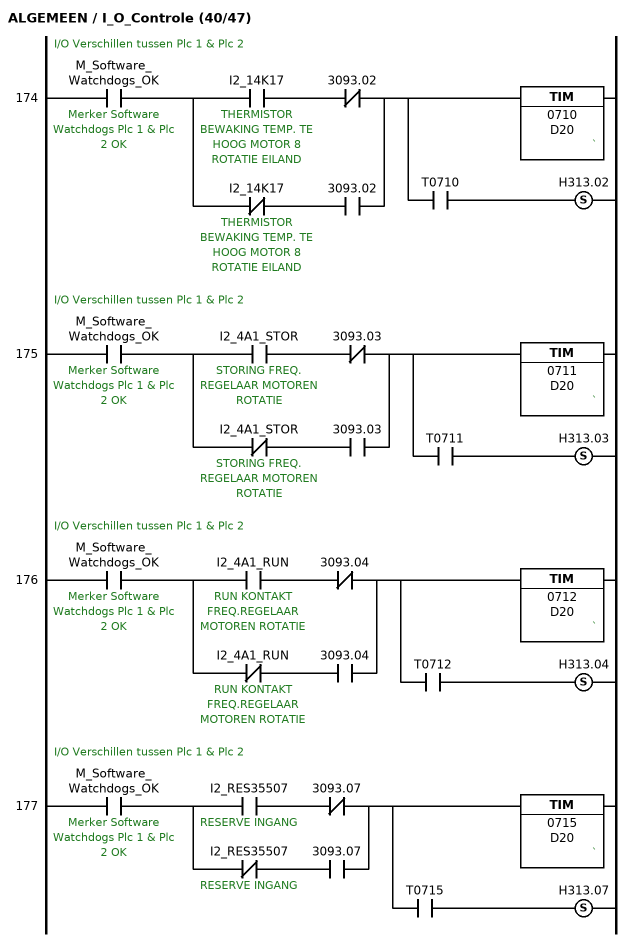
; rung 174: I/O Verschillen tussen Plc 1 & Plc 2
LD M_Software_Watchdogs_OK  ; Merker Software Watchdogs Plc 1 & Plc 2 OK
LD I2_14K17  ; THERMISTOR BEWAKING TEMP. TE HOOG MOTOR 8 ROTATIE EILAND
ANDNOT 3093.02
LDNOT I2_14K17  ; THERMISTOR BEWAKING TEMP. TE HOOG MOTOR 8 ROTATIE EILAND
AND 3093.02
ORLD
ANDLD
TIM 0710 D20  ; `
AND T0710
SET H313.02
; rung 175: I/O Verschillen tussen Plc 1 & Plc 2
LD M_Software_Watchdogs_OK  ; Merker Software Watchdogs Plc 1 & Plc 2 OK
LD I2_4A1_STOR  ; STORING FREQ.REGELAAR MOTOREN ROTATIE
ANDNOT 3093.03
LDNOT I2_4A1_STOR  ; STORING FREQ.REGELAAR MOTOREN ROTATIE
AND 3093.03
ORLD
ANDLD
TIM 0711 D20  ; `
AND T0711
SET H313.03
; rung 176: I/O Verschillen tussen Plc 1 & Plc 2
LD M_Software_Watchdogs_OK  ; Merker Software Watchdogs Plc 1 & Plc 2 OK
LD I2_4A1_RUN  ; RUN KONTAKT FREQ.REGELAAR MOTOREN ROTATIE
ANDNOT 3093.04
LDNOT I2_4A1_RUN  ; RUN KONTAKT FREQ.REGELAAR MOTOREN ROTATIE
AND 3093.04
ORLD
ANDLD
TIM 0712 D20  ; `
AND T0712
SET H313.04
; rung 177: I/O Verschillen tussen Plc 1 & Plc 2
LD M_Software_Watchdogs_OK  ; Merker Software Watchdogs Plc 1 & Plc 2 OK
LD I2_RES35507  ; RESERVE INGANG
ANDNOT 3093.07
LDNOT I2_RES35507  ; RESERVE INGANG
AND 3093.07
ORLD
ANDLD
TIM 0715 D20  ; `
AND T0715
SET H313.07

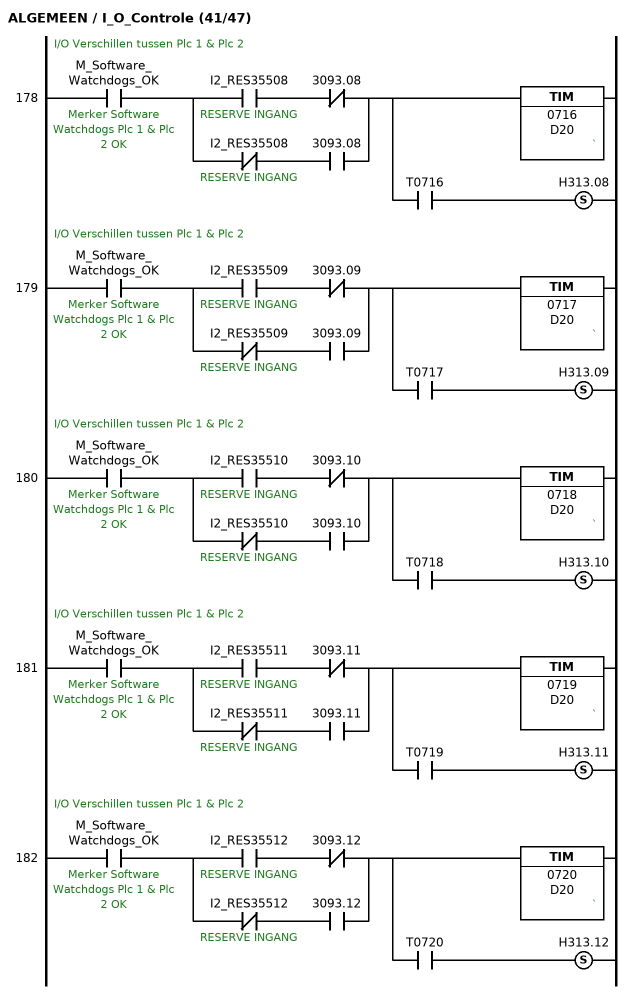
; rung 178: I/O Verschillen tussen Plc 1 & Plc 2
LD M_Software_Watchdogs_OK  ; Merker Software Watchdogs Plc 1 & Plc 2 OK
LD I2_RES35508  ; RESERVE INGANG
ANDNOT 3093.08
LDNOT I2_RES35508  ; RESERVE INGANG
AND 3093.08
ORLD
ANDLD
TIM 0716 D20  ; `
AND T0716
SET H313.08
; rung 179: I/O Verschillen tussen Plc 1 & Plc 2
LD M_Software_Watchdogs_OK  ; Merker Software Watchdogs Plc 1 & Plc 2 OK
LD I2_RES35509  ; RESERVE INGANG
ANDNOT 3093.09
LDNOT I2_RES35509  ; RESERVE INGANG
AND 3093.09
ORLD
ANDLD
TIM 0717 D20  ; `
AND T0717
SET H313.09
; rung 180: I/O Verschillen tussen Plc 1 & Plc 2
LD M_Software_Watchdogs_OK  ; Merker Software Watchdogs Plc 1 & Plc 2 OK
LD I2_RES35510  ; RESERVE INGANG
ANDNOT 3093.10
LDNOT I2_RES35510  ; RESERVE INGANG
AND 3093.10
ORLD
ANDLD
TIM 0718 D20  ; `
AND T0718
SET H313.10
; rung 181: I/O Verschillen tussen Plc 1 & Plc 2
LD M_Software_Watchdogs_OK  ; Merker Software Watchdogs Plc 1 & Plc 2 OK
LD I2_RES35511  ; RESERVE INGANG
ANDNOT 3093.11
LDNOT I2_RES35511  ; RESERVE INGANG
AND 3093.11
ORLD
ANDLD
TIM 0719 D20  ; `
AND T0719
SET H313.11
; rung 182: I/O Verschillen tussen Plc 1 & Plc 2
LD M_Software_Watchdogs_OK  ; Merker Software Watchdogs Plc 1 & Plc 2 OK
LD I2_RES35512  ; RESERVE INGANG
ANDNOT 3093.12
LDNOT I2_RES35512  ; RESERVE INGANG
AND 3093.12
ORLD
ANDLD
TIM 0720 D20  ; `
AND T0720
SET H313.12

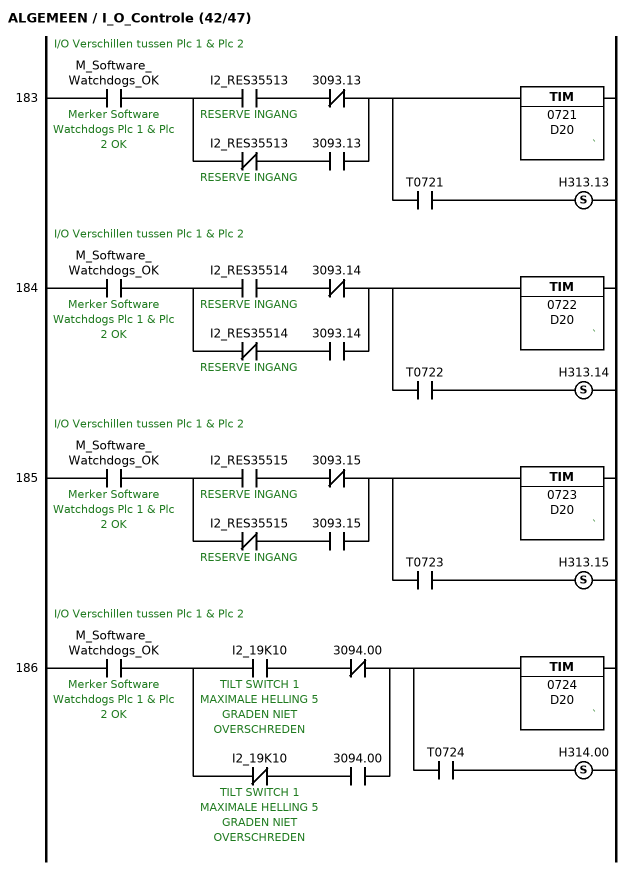
; rung 183: I/O Verschillen tussen Plc 1 & Plc 2
LD M_Software_Watchdogs_OK  ; Merker Software Watchdogs Plc 1 & Plc 2 OK
LD I2_RES35513  ; RESERVE INGANG
ANDNOT 3093.13
LDNOT I2_RES35513  ; RESERVE INGANG
AND 3093.13
ORLD
ANDLD
TIM 0721 D20  ; `
AND T0721
SET H313.13
; rung 184: I/O Verschillen tussen Plc 1 & Plc 2
LD M_Software_Watchdogs_OK  ; Merker Software Watchdogs Plc 1 & Plc 2 OK
LD I2_RES35514  ; RESERVE INGANG
ANDNOT 3093.14
LDNOT I2_RES35514  ; RESERVE INGANG
AND 3093.14
ORLD
ANDLD
TIM 0722 D20  ; `
AND T0722
SET H313.14
; rung 185: I/O Verschillen tussen Plc 1 & Plc 2
LD M_Software_Watchdogs_OK  ; Merker Software Watchdogs Plc 1 & Plc 2 OK
LD I2_RES35515  ; RESERVE INGANG
ANDNOT 3093.15
LDNOT I2_RES35515  ; RESERVE INGANG
AND 3093.15
ORLD
ANDLD
TIM 0723 D20  ; `
AND T0723
SET H313.15
; rung 186: I/O Verschillen tussen Plc 1 & Plc 2
LD M_Software_Watchdogs_OK  ; Merker Software Watchdogs Plc 1 & Plc 2 OK
LD I2_19K10  ; TILT SWITCH 1 MAXIMALE HELLING 5 GRADEN NIET OVERSCHREDEN
ANDNOT 3094.00
LDNOT I2_19K10  ; TILT SWITCH 1 MAXIMALE HELLING 5 GRADEN NIET OVERSCHREDEN
AND 3094.00
ORLD
ANDLD
TIM 0724 D20  ; `
AND T0724
SET H314.00

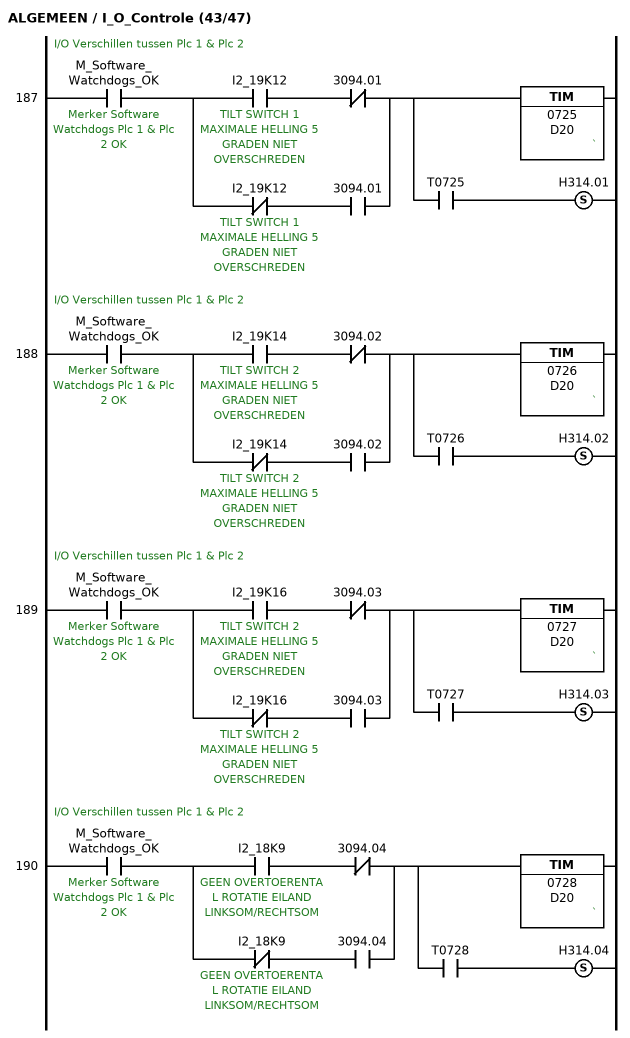
; rung 187: I/O Verschillen tussen Plc 1 & Plc 2
LD M_Software_Watchdogs_OK  ; Merker Software Watchdogs Plc 1 & Plc 2 OK
LD I2_19K12  ; TILT SWITCH 1 MAXIMALE HELLING 5 GRADEN NIET OVERSCHREDEN
ANDNOT 3094.01
LDNOT I2_19K12  ; TILT SWITCH 1 MAXIMALE HELLING 5 GRADEN NIET OVERSCHREDEN
AND 3094.01
ORLD
ANDLD
TIM 0725 D20  ; `
AND T0725
SET H314.01
; rung 188: I/O Verschillen tussen Plc 1 & Plc 2
LD M_Software_Watchdogs_OK  ; Merker Software Watchdogs Plc 1 & Plc 2 OK
LD I2_19K14  ; TILT SWITCH 2 MAXIMALE HELLING 5 GRADEN NIET OVERSCHREDEN
ANDNOT 3094.02
LDNOT I2_19K14  ; TILT SWITCH 2 MAXIMALE HELLING 5 GRADEN NIET OVERSCHREDEN
AND 3094.02
ORLD
ANDLD
TIM 0726 D20  ; `
AND T0726
SET H314.02
; rung 189: I/O Verschillen tussen Plc 1 & Plc 2
LD M_Software_Watchdogs_OK  ; Merker Software Watchdogs Plc 1 & Plc 2 OK
LD I2_19K16  ; TILT SWITCH 2 MAXIMALE HELLING 5 GRADEN NIET OVERSCHREDEN
ANDNOT 3094.03
LDNOT I2_19K16  ; TILT SWITCH 2 MAXIMALE HELLING 5 GRADEN NIET OVERSCHREDEN
AND 3094.03
ORLD
ANDLD
TIM 0727 D20  ; `
AND T0727
SET H314.03
; rung 190: I/O Verschillen tussen Plc 1 & Plc 2
LD M_Software_Watchdogs_OK  ; Merker Software Watchdogs Plc 1 & Plc 2 OK
LD I2_18K9  ; GEEN OVERTOERENTAL ROTATIE EILAND LINKSOM/RECHTSOM
ANDNOT 3094.04
LDNOT I2_18K9  ; GEEN OVERTOERENTAL ROTATIE EILAND LINKSOM/RECHTSOM
AND 3094.04
ORLD
ANDLD
TIM 0728 D20  ; `
AND T0728
SET H314.04

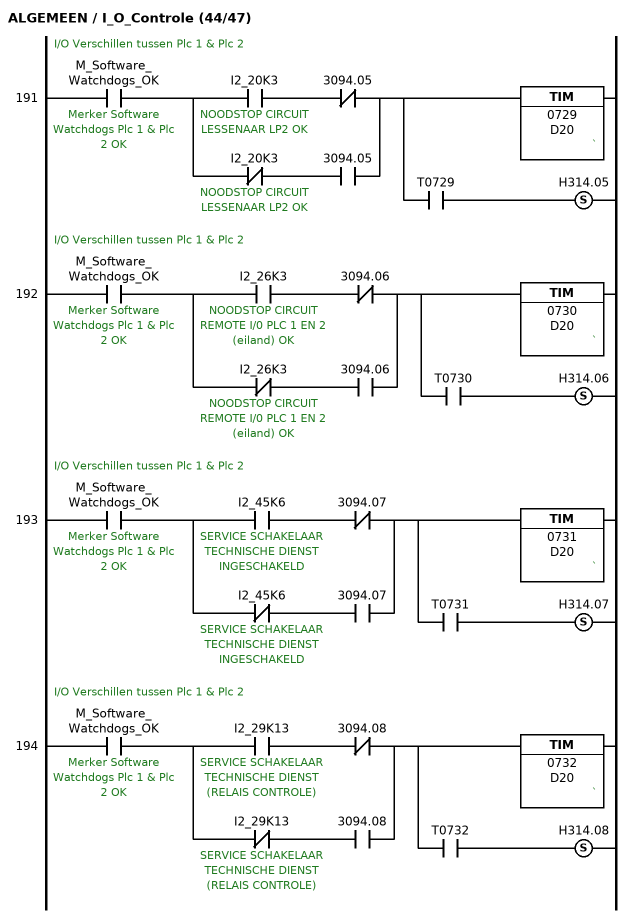
; rung 191: I/O Verschillen tussen Plc 1 & Plc 2
LD M_Software_Watchdogs_OK  ; Merker Software Watchdogs Plc 1 & Plc 2 OK
LD I2_20K3  ; NOODSTOP CIRCUIT LESSENAAR LP2 OK
ANDNOT 3094.05
LDNOT I2_20K3  ; NOODSTOP CIRCUIT LESSENAAR LP2 OK
AND 3094.05
ORLD
ANDLD
TIM 0729 D20  ; `
AND T0729
SET H314.05
; rung 192: I/O Verschillen tussen Plc 1 & Plc 2
LD M_Software_Watchdogs_OK  ; Merker Software Watchdogs Plc 1 & Plc 2 OK
LD I2_26K3  ; NOODSTOP CIRCUIT REMOTE I/0 PLC 1 EN 2 (eiland) OK
ANDNOT 3094.06
LDNOT I2_26K3  ; NOODSTOP CIRCUIT REMOTE I/0 PLC 1 EN 2 (eiland) OK
AND 3094.06
ORLD
ANDLD
TIM 0730 D20  ; `
AND T0730
SET H314.06
; rung 193: I/O Verschillen tussen Plc 1 & Plc 2
LD M_Software_Watchdogs_OK  ; Merker Software Watchdogs Plc 1 & Plc 2 OK
LD I2_45K6  ; SERVICE SCHAKELAAR TECHNISCHE DIENST INGESCHAKELD
ANDNOT 3094.07
LDNOT I2_45K6  ; SERVICE SCHAKELAAR TECHNISCHE DIENST INGESCHAKELD
AND 3094.07
ORLD
ANDLD
TIM 0731 D20  ; `
AND T0731
SET H314.07
; rung 194: I/O Verschillen tussen Plc 1 & Plc 2
LD M_Software_Watchdogs_OK  ; Merker Software Watchdogs Plc 1 & Plc 2 OK
LD I2_29K13  ; SERVICE SCHAKELAAR TECHNISCHE DIENST (RELAIS CONTROLE)
ANDNOT 3094.08
LDNOT I2_29K13  ; SERVICE SCHAKELAAR TECHNISCHE DIENST (RELAIS CONTROLE)
AND 3094.08
ORLD
ANDLD
TIM 0732 D20  ; `
AND T0732
SET H314.08

